   BB2_AS2.Stoerung.Res_24 := FALSE;
   BB2_AS2.Stoerung.Res_25 := FALSE;
   BB2_AS2.Stoerung.Res_26 := FALSE;
   BB2_AS2.Stoerung.Res_27 := FALSE;
   BB2_AS2.Stoerung.Res_28 := FALSE;
   BB2_AS2.Stoerung.Res_29 := FALSE;
   BB2_AS2.Stoerung.Res_30 := FALSE;
   BB2_AS2.Stoerung.Res_31 := FALSE;
   BB2_AS2.MW_I := 0.0;
   BB2_AS2.MW_P := 0.0;
   BB2_AS2.EZ := 0;
   BB2_AS2.BZ_akt := 27;
   BB2_AS2.BZ_ges := 978766;
   BB2_AS2.AZ_akt := 2137;
   BB2_AS2.ESH := 35306;
   BB2_AS2.SW_akt := 0.0;
   BB2_AS2.SW_Auto := 0.0;
   BB2_AS2.SW_out := 0.0;
   BB2_SR1.Status.Bed_vOrt := FALSE;
   BB2_SR1.Status.Bed_UV := FALSE;
   BB2_SR1.Status.Bed_NHV := FALSE;
   BB2_SR1.Status.Bed_PLS := TRUE;
   BB2_SR1.Status.BA_Hand := FALSE;
   BB2_SR1.Status.BA_Auto := TRUE;
   BB2_SR1.Status.RB_Ein1 := FALSE;
   BB2_SR1.Status.RB_Ein2 := FALSE;
   BB2_SR1.Status.RB_Aus := TRUE;
   BB2_SR1.Status.BFR_NS := FALSE;
   BB2_SR1.Status.BFR_ECS := FALSE;
   BB2_SR1.Status.BFR_ESK := FALSE;
   BB2_SR1.Status.BFR_MAZ := FALSE;
   BB2_SR1.Status.BFR_Rev := FALSE;
   BB2_SR1.Status.BFR_Ein1 := FALSE;
   BB2_SR1.Status.BFR_Ein2 := FALSE;
   BB2_SR1.Status.BM_Ein1 := FALSE;
   BB2_SR1.Status.BM_Ein2 := FALSE;
   BB2_SR1.Status.BM_Auf := FALSE;
   BB2_SR1.Status.BM_Zu := TRUE;
   BB2_SR1.Status.BM_Ein := FALSE;
   BB2_SR1.Status.BM_Aus := TRUE;
   BB2_SR1.Status.BM_Anst1 := FALSE;
   BB2_SR1.Status.BM_Anst2 := FALSE;
   BB2_SR1.Status.BM_Auto1 := FALSE;
   BB2_SR1.Status.BM_Auto2 := TRUE;
   BB2_SR1.Status.Res_26 := FALSE;
   BB2_SR1.Status.Res_27 := FALSE;
   BB2_SR1.Status.BB_NA := FALSE;
   BB2_SR1.Status.BB_AutoOk := TRUE;
   BB2_SR1.Status.BB_SS := FALSE;
   BB2_SR1.Status.BB_SSnq := FALSE;
   BB2_SR1.Stoerung.St_allg := FALSE;
   BB2_SR1.Stoerung.St_DMA := FALSE;
   BB2_SR1.Stoerung.St_DMZ := FALSE;
   BB2_SR1.Stoerung.St_FU := FALSE;
   BB2_SR1.Stoerung.St_TL := FALSE;
   BB2_SR1.Stoerung.St_UDr := FALSE;
   BB2_SR1.Stoerung.St_UeDr := FALSE;
   BB2_SR1.Stoerung.St_UeTemp := FALSE;
   BB2_SR1.Stoerung.St_Leck := FALSE;
   BB2_SR1.Stoerung.St_UeLM := FALSE;
   BB2_SR1.Stoerung.St_UeLE := FALSE;
   BB2_SR1.Stoerung.St_Kom_DP := FALSE;
   BB2_SR1.Stoerung.St_Kom_int := FALSE;
   BB2_SR1.Stoerung.St_int := FALSE;
   BB2_SR1.Stoerung.St_LZ := FALSE;
   BB2_SR1.Stoerung.St_BefLZ := FALSE;
   BB2_SR1.Stoerung.Wa_EZ := FALSE;
   BB2_SR1.Stoerung.Wa_Wart := FALSE;
   BB2_SR1.Stoerung.St_Strm := FALSE;
   BB2_SR1.Stoerung.Res_19 := FALSE;
   BB2_SR1.Stoerung.Res_20 := FALSE;
   BB2_SR1.Stoerung.Res_21 := FALSE;
   BB2_SR1.Stoerung.Res_22 := FALSE;
   BB2_SR1.Stoerung.Res_23 := FALSE;
   BB2_SR1.Stoerung.Res_24 := FALSE;
   BB2_SR1.Stoerung.Res_25 := FALSE;
   BB2_SR1.Stoerung.Res_26 := FALSE;
   BB2_SR1.Stoerung.Res_27 := FALSE;
   BB2_SR1.Stoerung.Res_28 := FALSE;
   BB2_SR1.Stoerung.Res_29 := FALSE;
   BB2_SR1.Stoerung.Res_30 := FALSE;
   BB2_SR1.Stoerung.Res_31 := FALSE;
   BB2_SR1.MW_I := 0.0;
   BB2_SR1.MW_P := 0.0;
   BB2_SR1.EZ := 0;
   BB2_SR1.BZ_akt := 179;
   BB2_SR1.BZ_ges := 3159816;
   BB2_SR1.AZ_akt := 5585;
   BB2_SR1.ESH := 17588;
   BB2_SR1.SW_akt := 0.0;
   BB2_SR1.SW_Auto := 0.0;
   BB2_SR1.SW_out := 0.0;
   BB2_SR2.Status.Bed_vOrt := FALSE;
   BB2_SR2.Status.Bed_UV := FALSE;
   BB2_SR2.Status.Bed_NHV := FALSE;
   BB2_SR2.Status.Bed_PLS := TRUE;
   BB2_SR2.Status.BA_Hand := FALSE;
   BB2_SR2.Status.BA_Auto := TRUE;
   BB2_SR2.Status.RB_Ein1 := FALSE;
   BB2_SR2.Status.RB_Ein2 := FALSE;
   BB2_SR2.Status.RB_Aus := TRUE;
   BB2_SR2.Status.BFR_NS := FALSE;
   BB2_SR2.Status.BFR_ECS := FALSE;
   BB2_SR2.Status.BFR_ESK := FALSE;
   BB2_SR2.Status.BFR_MAZ := FALSE;
   BB2_SR2.Status.BFR_Rev := FALSE;
   BB2_SR2.Status.BFR_Ein1 := FALSE;
   BB2_SR2.Status.BFR_Ein2 := FALSE;
   BB2_SR2.Status.BM_Ein1 := FALSE;
   BB2_SR2.Status.BM_Ein2 := FALSE;
   BB2_SR2.Status.BM_Auf := FALSE;
   BB2_SR2.Status.BM_Zu := TRUE;
   BB2_SR2.Status.BM_Ein := FALSE;
   BB2_SR2.Status.BM_Aus := TRUE;
   BB2_SR2.Status.BM_Anst1 := FALSE;
   BB2_SR2.Status.BM_Anst2 := FALSE;
   BB2_SR2.Status.BM_Auto1 := FALSE;
   BB2_SR2.Status.BM_Auto2 := TRUE;
   BB2_SR2.Status.Res_26 := FALSE;
   BB2_SR2.Status.Res_27 := FALSE;
   BB2_SR2.Status.BB_NA := FALSE;
   BB2_SR2.Status.BB_AutoOk := TRUE;
   BB2_SR2.Status.BB_SS := FALSE;
   BB2_SR2.Status.BB_SSnq := FALSE;
   BB2_SR2.Stoerung.St_allg := FALSE;
   BB2_SR2.Stoerung.St_DMA := FALSE;
   BB2_SR2.Stoerung.St_DMZ := FALSE;
   BB2_SR2.Stoerung.St_FU := FALSE;
   BB2_SR2.Stoerung.St_TL := FALSE;
   BB2_SR2.Stoerung.St_UDr := FALSE;
   BB2_SR2.Stoerung.St_UeDr := FALSE;
   BB2_SR2.Stoerung.St_UeTemp := FALSE;
   BB2_SR2.Stoerung.St_Leck := FALSE;
   BB2_SR2.Stoerung.St_UeLM := FALSE;
   BB2_SR2.Stoerung.St_UeLE := FALSE;
   BB2_SR2.Stoerung.St_Kom_DP := FALSE;
   BB2_SR2.Stoerung.St_Kom_int := FALSE;
   BB2_SR2.Stoerung.St_int := FALSE;
   BB2_SR2.Stoerung.St_LZ := FALSE;
   BB2_SR2.Stoerung.St_BefLZ := FALSE;
   BB2_SR2.Stoerung.Wa_EZ := FALSE;
   BB2_SR2.Stoerung.Wa_Wart := FALSE;
   BB2_SR2.Stoerung.St_Strm := FALSE;
   BB2_SR2.Stoerung.Res_19 := FALSE;
   BB2_SR2.Stoerung.Res_20 := FALSE;
   BB2_SR2.Stoerung.Res_21 := FALSE;
   BB2_SR2.Stoerung.Res_22 := FALSE;
   BB2_SR2.Stoerung.Res_23 := FALSE;
   BB2_SR2.Stoerung.Res_24 := FALSE;
   BB2_SR2.Stoerung.Res_25 := FALSE;
   BB2_SR2.Stoerung.Res_26 := FALSE;
   BB2_SR2.Stoerung.Res_27 := FALSE;
   BB2_SR2.Stoerung.Res_28 := FALSE;
   BB2_SR2.Stoerung.Res_29 := FALSE;
   BB2_SR2.Stoerung.Res_30 := FALSE;
   BB2_SR2.Stoerung.Res_31 := FALSE;
   BB2_SR2.MW_I := 0.0;
   BB2_SR2.MW_P := 0.0;
   BB2_SR2.EZ := 0;
   BB2_SR2.BZ_akt := 179;
   BB2_SR2.BZ_ges := 3129764;
   BB2_SR2.AZ_akt := 1985;
   BB2_SR2.ESH := 17409;
   BB2_SR2.SW_akt := 0.0;
   BB2_SR2.SW_Auto := 0.0;
   BB2_SR2.SW_out := 0.0;
   BB1_SR_K.Status.Bed_vOrt := FALSE;
   BB1_SR_K.Status.Bed_UV := FALSE;
   BB1_SR_K.Status.Bed_NHV := TRUE;
   BB1_SR_K.Status.Bed_PLS := FALSE;
   BB1_SR_K.Status.BA_Hand := FALSE;
   BB1_SR_K.Status.BA_Auto := TRUE;
   BB1_SR_K.Status.RB_Ein1 := FALSE;
   BB1_SR_K.Status.RB_Ein2 := FALSE;
   BB1_SR_K.Status.RB_Aus := TRUE;
   BB1_SR_K.Status.BFR_NS := FALSE;
   BB1_SR_K.Status.BFR_ECS := FALSE;
   BB1_SR_K.Status.BFR_ESK := FALSE;
   BB1_SR_K.Status.BFR_MAZ := FALSE;
   BB1_SR_K.Status.BFR_Rev := FALSE;
   BB1_SR_K.Status.BFR_Ein1 := FALSE;
   BB1_SR_K.Status.BFR_Ein2 := FALSE;
   BB1_SR_K.Status.BM_Ein1 := FALSE;
   BB1_SR_K.Status.BM_Ein2 := FALSE;
   BB1_SR_K.Status.BM_Auf := FALSE;
   BB1_SR_K.Status.BM_Zu := FALSE;
   BB1_SR_K.Status.BM_Ein := FALSE;
   BB1_SR_K.Status.BM_Aus := TRUE;
   BB1_SR_K.Status.BM_Anst1 := FALSE;
   BB1_SR_K.Status.BM_Anst2 := FALSE;
   BB1_SR_K.Status.BM_Auto1 := FALSE;
   BB1_SR_K.Status.BM_Auto2 := FALSE;
   BB1_SR_K.Status.Res_26 := FALSE;
   BB1_SR_K.Status.Res_27 := FALSE;
   BB1_SR_K.Status.BB_NA := FALSE;
   BB1_SR_K.Status.BB_AutoOk := FALSE;
   BB1_SR_K.Status.BB_SS := TRUE;
   BB1_SR_K.Status.BB_SSnq := FALSE;
   BB1_SR_K.Stoerung.St_allg := TRUE;
   BB1_SR_K.Stoerung.St_DMA := FALSE;
   BB1_SR_K.Stoerung.St_DMZ := FALSE;
   BB1_SR_K.Stoerung.St_FU := FALSE;
   BB1_SR_K.Stoerung.St_TL := FALSE;
   BB1_SR_K.Stoerung.St_UDr := FALSE;
   BB1_SR_K.Stoerung.St_UeDr := FALSE;
   BB1_SR_K.Stoerung.St_UeTemp := FALSE;
   BB1_SR_K.Stoerung.St_Leck := FALSE;
   BB1_SR_K.Stoerung.St_UeLM := FALSE;
   BB1_SR_K.Stoerung.St_UeLE := FALSE;
   BB1_SR_K.Stoerung.St_Kom_DP := FALSE;
   BB1_SR_K.Stoerung.St_Kom_int := FALSE;
   BB1_SR_K.Stoerung.St_int := FALSE;
   BB1_SR_K.Stoerung.St_LZ := FALSE;
   BB1_SR_K.Stoerung.St_BefLZ := FALSE;
   BB1_SR_K.Stoerung.Wa_EZ := FALSE;
   BB1_SR_K.Stoerung.Wa_Wart := FALSE;
   BB1_SR_K.Stoerung.St_Strm := FALSE;
   BB1_SR_K.Stoerung.Res_19 := FALSE;
   BB1_SR_K.Stoerung.Res_20 := FALSE;
   BB1_SR_K.Stoerung.Res_21 := FALSE;
   BB1_SR_K.Stoerung.Res_22 := FALSE;
   BB1_SR_K.Stoerung.Res_23 := FALSE;
   BB1_SR_K.Stoerung.Res_24 := FALSE;
   BB1_SR_K.Stoerung.Res_25 := FALSE;
   BB1_SR_K.Stoerung.Res_26 := FALSE;
   BB1_SR_K.Stoerung.Res_27 := FALSE;
   BB1_SR_K.Stoerung.Res_28 := FALSE;
   BB1_SR_K.Stoerung.Res_29 := FALSE;
   BB1_SR_K.Stoerung.Res_30 := FALSE;
   BB1_SR_K.Stoerung.Res_31 := FALSE;
   BB1_SR_K.MW_I := 0.0;
   BB1_SR_K.MW_P := 0.0;
   BB1_SR_K.EZ := 0;
   BB1_SR_K.BZ_akt := 180;
   BB1_SR_K.BZ_ges := 6365850;
   BB1_SR_K.AZ_akt := 2005;
   BB1_SR_K.ESH := 34998;
   BB1_SR_K.SW_akt := 0.0;
   BB1_SR_K.SW_Auto := 0.0;
   BB1_SR_K.SW_out := 0.0;
   Zulauf_AR_P1.Status.Bed_vOrt := FALSE;
   Zulauf_AR_P1.Status.Bed_UV := FALSE;
   Zulauf_AR_P1.Status.Bed_NHV := TRUE;
   Zulauf_AR_P1.Status.Bed_PLS := FALSE;
   Zulauf_AR_P1.Status.BA_Hand := FALSE;
   Zulauf_AR_P1.Status.BA_Auto := TRUE;
   Zulauf_AR_P1.Status.RB_Ein1 := FALSE;
   Zulauf_AR_P1.Status.RB_Ein2 := FALSE;
   Zulauf_AR_P1.Status.RB_Aus := TRUE;
   Zulauf_AR_P1.Status.BFR_NS := FALSE;
   Zulauf_AR_P1.Status.BFR_ECS := FALSE;
   Zulauf_AR_P1.Status.BFR_ESK := FALSE;
   Zulauf_AR_P1.Status.BFR_MAZ := FALSE;
   Zulauf_AR_P1.Status.BFR_Rev := FALSE;
   Zulauf_AR_P1.Status.BFR_Ein1 := FALSE;
   Zulauf_AR_P1.Status.BFR_Ein2 := FALSE;
   Zulauf_AR_P1.Status.BM_Ein1 := FALSE;
   Zulauf_AR_P1.Status.BM_Ein2 := FALSE;
   Zulauf_AR_P1.Status.BM_Auf := FALSE;
   Zulauf_AR_P1.Status.BM_Zu := FALSE;
   Zulauf_AR_P1.Status.BM_Ein := FALSE;
   Zulauf_AR_P1.Status.BM_Aus := TRUE;
   Zulauf_AR_P1.Status.BM_Anst1 := FALSE;
   Zulauf_AR_P1.Status.BM_Anst2 := FALSE;
   Zulauf_AR_P1.Status.BM_Auto1 := FALSE;
   Zulauf_AR_P1.Status.BM_Auto2 := FALSE;
   Zulauf_AR_P1.Status.Res_26 := FALSE;
   Zulauf_AR_P1.Status.Res_27 := FALSE;
   Zulauf_AR_P1.Status.BB_NA := FALSE;
   Zulauf_AR_P1.Status.BB_AutoOk := TRUE;
   Zulauf_AR_P1.Status.BB_SS := FALSE;
   Zulauf_AR_P1.Status.BB_SSnq := FALSE;
   Zulauf_AR_P1.Stoerung.St_allg := FALSE;
   Zulauf_AR_P1.Stoerung.St_DMA := FALSE;
   Zulauf_AR_P1.Stoerung.St_DMZ := FALSE;
   Zulauf_AR_P1.Stoerung.St_FU := FALSE;
   Zulauf_AR_P1.Stoerung.St_TL := FALSE;
   Zulauf_AR_P1.Stoerung.St_UDr := FALSE;
   Zulauf_AR_P1.Stoerung.St_UeDr := FALSE;
   Zulauf_AR_P1.Stoerung.St_UeTemp := FALSE;
   Zulauf_AR_P1.Stoerung.St_Leck := FALSE;
   Zulauf_AR_P1.Stoerung.St_UeLM := FALSE;
   Zulauf_AR_P1.Stoerung.St_UeLE := FALSE;
   Zulauf_AR_P1.Stoerung.St_Kom_DP := FALSE;
   Zulauf_AR_P1.Stoerung.St_Kom_int := FALSE;
   Zulauf_AR_P1.Stoerung.St_int := FALSE;
   Zulauf_AR_P1.Stoerung.St_LZ := FALSE;
   Zulauf_AR_P1.Stoerung.St_BefLZ := FALSE;
   Zulauf_AR_P1.Stoerung.Wa_EZ := FALSE;
   Zulauf_AR_P1.Stoerung.Wa_Wart := FALSE;
   Zulauf_AR_P1.Stoerung.St_Strm := FALSE;
   Zulauf_AR_P1.Stoerung.Res_19 := FALSE;
   Zulauf_AR_P1.Stoerung.Res_20 := FALSE;
   Zulauf_AR_P1.Stoerung.Res_21 := FALSE;
   Zulauf_AR_P1.Stoerung.Res_22 := FALSE;
   Zulauf_AR_P1.Stoerung.Res_23 := FALSE;
   Zulauf_AR_P1.Stoerung.Res_24 := FALSE;
   Zulauf_AR_P1.Stoerung.Res_25 := FALSE;
   Zulauf_AR_P1.Stoerung.Res_26 := FALSE;
   Zulauf_AR_P1.Stoerung.Res_27 := FALSE;
   Zulauf_AR_P1.Stoerung.Res_28 := FALSE;
   Zulauf_AR_P1.Stoerung.Res_29 := FALSE;
   Zulauf_AR_P1.Stoerung.Res_30 := FALSE;
   Zulauf_AR_P1.Stoerung.Res_31 := FALSE;
   Zulauf_AR_P1.MW_I := 0.0;
   Zulauf_AR_P1.MW_P := 0.0;
   Zulauf_AR_P1.EZ := 0;
   Zulauf_AR_P1.BZ_akt := 0;
   Zulauf_AR_P1.BZ_ges := 0;
   Zulauf_AR_P1.AZ_akt := 132_442_977;
   Zulauf_AR_P1.ESH := 0;
   Zulauf_AR_P1.SW_akt := 0.0;
   Zulauf_AR_P1.SW_Auto := 0.0;
   Zulauf_AR_P1.SW_out := 0.0;
   Zulauf_AR_P2.Status.Bed_vOrt := FALSE;
   Zulauf_AR_P2.Status.Bed_UV := FALSE;
   Zulauf_AR_P2.Status.Bed_NHV := TRUE;
   Zulauf_AR_P2.Status.Bed_PLS := FALSE;
   Zulauf_AR_P2.Status.BA_Hand := FALSE;
   Zulauf_AR_P2.Status.BA_Auto := TRUE;
   Zulauf_AR_P2.Status.RB_Ein1 := FALSE;
   Zulauf_AR_P2.Status.RB_Ein2 := FALSE;
   Zulauf_AR_P2.Status.RB_Aus := TRUE;
   Zulauf_AR_P2.Status.BFR_NS := FALSE;
   Zulauf_AR_P2.Status.BFR_ECS := FALSE;
   Zulauf_AR_P2.Status.BFR_ESK := FALSE;
   Zulauf_AR_P2.Status.BFR_MAZ := FALSE;
   Zulauf_AR_P2.Status.BFR_Rev := FALSE;
   Zulauf_AR_P2.Status.BFR_Ein1 := FALSE;
   Zulauf_AR_P2.Status.BFR_Ein2 := FALSE;
   Zulauf_AR_P2.Status.BM_Ein1 := FALSE;
   Zulauf_AR_P2.Status.BM_Ein2 := FALSE;
   Zulauf_AR_P2.Status.BM_Auf := FALSE;
   Zulauf_AR_P2.Status.BM_Zu := FALSE;
   Zulauf_AR_P2.Status.BM_Ein := FALSE;
   Zulauf_AR_P2.Status.BM_Aus := TRUE;
   Zulauf_AR_P2.Status.BM_Anst1 := FALSE;
   Zulauf_AR_P2.Status.BM_Anst2 := FALSE;
   Zulauf_AR_P2.Status.BM_Auto1 := FALSE;
   Zulauf_AR_P2.Status.BM_Auto2 := FALSE;
   Zulauf_AR_P2.Status.Res_26 := FALSE;
   Zulauf_AR_P2.Status.Res_27 := FALSE;
   Zulauf_AR_P2.Status.BB_NA := FALSE;
   Zulauf_AR_P2.Status.BB_AutoOk := TRUE;
   Zulauf_AR_P2.Status.BB_SS := FALSE;
   Zulauf_AR_P2.Status.BB_SSnq := FALSE;
   Zulauf_AR_P2.Stoerung.St_allg := FALSE;
   Zulauf_AR_P2.Stoerung.St_DMA := FALSE;
   Zulauf_AR_P2.Stoerung.St_DMZ := FALSE;
   Zulauf_AR_P2.Stoerung.St_FU := FALSE;
   Zulauf_AR_P2.Stoerung.St_TL := FALSE;
   Zulauf_AR_P2.Stoerung.St_UDr := FALSE;
   Zulauf_AR_P2.Stoerung.St_UeDr := FALSE;
   Zulauf_AR_P2.Stoerung.St_UeTemp := FALSE;
   Zulauf_AR_P2.Stoerung.St_Leck := FALSE;
   Zulauf_AR_P2.Stoerung.St_UeLM := FALSE;
   Zulauf_AR_P2.Stoerung.St_UeLE := FALSE;
   Zulauf_AR_P2.Stoerung.St_Kom_DP := FALSE;
   Zulauf_AR_P2.Stoerung.St_Kom_int := FALSE;
   Zulauf_AR_P2.Stoerung.St_int := FALSE;
   Zulauf_AR_P2.Stoerung.St_LZ := FALSE;
   Zulauf_AR_P2.Stoerung.St_BefLZ := FALSE;
   Zulauf_AR_P2.Stoerung.Wa_EZ := FALSE;
   Zulauf_AR_P2.Stoerung.Wa_Wart := FALSE;
   Zulauf_AR_P2.Stoerung.St_Strm := FALSE;
   Zulauf_AR_P2.Stoerung.Res_19 := FALSE;
   Zulauf_AR_P2.Stoerung.Res_20 := FALSE;
   Zulauf_AR_P2.Stoerung.Res_21 := FALSE;
   Zulauf_AR_P2.Stoerung.Res_22 := FALSE;
   Zulauf_AR_P2.Stoerung.Res_23 := FALSE;
   Zulauf_AR_P2.Stoerung.Res_24 := FALSE;
   Zulauf_AR_P2.Stoerung.Res_25 := FALSE;
   Zulauf_AR_P2.Stoerung.Res_26 := FALSE;
   Zulauf_AR_P2.Stoerung.Res_27 := FALSE;
   Zulauf_AR_P2.Stoerung.Res_28 := FALSE;
   Zulauf_AR_P2.Stoerung.Res_29 := FALSE;
   Zulauf_AR_P2.Stoerung.Res_30 := FALSE;
   Zulauf_AR_P2.Stoerung.Res_31 := FALSE;
   Zulauf_AR_P2.MW_I := 0.0;
   Zulauf_AR_P2.MW_P := 0.0;
   Zulauf_AR_P2.EZ := 0;
   Zulauf_AR_P2.BZ_akt := 676;
   Zulauf_AR_P2.BZ_ges := 676;
   Zulauf_AR_P2.AZ_akt := 132_196_371;
   Zulauf_AR_P2.ESH := 1;
   Zulauf_AR_P2.SW_akt := 0.0;
   Zulauf_AR_P2.SW_Auto := 0.0;
   Zulauf_AR_P2.SW_out := 0.0;
   Zulauf_AS.Status.Bed_vOrt := FALSE;
   Zulauf_AS.Status.Bed_UV := FALSE;
   Zulauf_AS.Status.Bed_NHV := TRUE;
   Zulauf_AS.Status.Bed_PLS := FALSE;
   Zulauf_AS.Status.BA_Hand := FALSE;
   Zulauf_AS.Status.BA_Auto := TRUE;
   Zulauf_AS.Status.RB_Ein1 := FALSE;
   Zulauf_AS.Status.RB_Ein2 := FALSE;
   Zulauf_AS.Status.RB_Aus := TRUE;
   Zulauf_AS.Status.BFR_NS := FALSE;
   Zulauf_AS.Status.BFR_ECS := FALSE;
   Zulauf_AS.Status.BFR_ESK := FALSE;
   Zulauf_AS.Status.BFR_MAZ := FALSE;
   Zulauf_AS.Status.BFR_Rev := FALSE;
   Zulauf_AS.Status.BFR_Ein1 := FALSE;
   Zulauf_AS.Status.BFR_Ein2 := FALSE;
   Zulauf_AS.Status.BM_Ein1 := FALSE;
   Zulauf_AS.Status.BM_Ein2 := FALSE;
   Zulauf_AS.Status.BM_Auf := FALSE;
   Zulauf_AS.Status.BM_Zu := FALSE;
   Zulauf_AS.Status.BM_Ein := FALSE;
   Zulauf_AS.Status.BM_Aus := TRUE;
   Zulauf_AS.Status.BM_Anst1 := FALSE;
   Zulauf_AS.Status.BM_Anst2 := FALSE;
   Zulauf_AS.Status.BM_Auto1 := FALSE;
   Zulauf_AS.Status.BM_Auto2 := FALSE;
   Zulauf_AS.Status.Res_26 := FALSE;
   Zulauf_AS.Status.Res_27 := FALSE;
   Zulauf_AS.Status.BB_NA := FALSE;
   Zulauf_AS.Status.BB_AutoOk := FALSE;
   Zulauf_AS.Status.BB_SS := TRUE;
   Zulauf_AS.Status.BB_SSnq := TRUE;
   Zulauf_AS.Stoerung.St_allg := TRUE;
   Zulauf_AS.Stoerung.St_DMA := FALSE;
   Zulauf_AS.Stoerung.St_DMZ := FALSE;
   Zulauf_AS.Stoerung.St_FU := FALSE;
   Zulauf_AS.Stoerung.St_TL := FALSE;
   Zulauf_AS.Stoerung.St_UDr := FALSE;
   Zulauf_AS.Stoerung.St_UeDr := FALSE;
   Zulauf_AS.Stoerung.St_UeTemp := FALSE;
   Zulauf_AS.Stoerung.St_Leck := FALSE;
   Zulauf_AS.Stoerung.St_UeLM := FALSE;
   Zulauf_AS.Stoerung.St_UeLE := FALSE;
   Zulauf_AS.Stoerung.St_Kom_DP := FALSE;
   Zulauf_AS.Stoerung.St_Kom_int := FALSE;
   Zulauf_AS.Stoerung.St_int := FALSE;
   Zulauf_AS.Stoerung.St_LZ := FALSE;
   Zulauf_AS.Stoerung.St_BefLZ := FALSE;
   Zulauf_AS.Stoerung.Wa_EZ := FALSE;
   Zulauf_AS.Stoerung.Wa_Wart := FALSE;
   Zulauf_AS.Stoerung.St_Strm := FALSE;
   Zulauf_AS.Stoerung.Res_19 := FALSE;
   Zulauf_AS.Stoerung.Res_20 := FALSE;
   Zulauf_AS.Stoerung.Res_21 := FALSE;
   Zulauf_AS.Stoerung.Res_22 := FALSE;
   Zulauf_AS.Stoerung.Res_23 := FALSE;
   Zulauf_AS.Stoerung.Res_24 := FALSE;
   Zulauf_AS.Stoerung.Res_25 := FALSE;
   Zulauf_AS.Stoerung.Res_26 := FALSE;
   Zulauf_AS.Stoerung.Res_27 := FALSE;
   Zulauf_AS.Stoerung.Res_28 := FALSE;
   Zulauf_AS.Stoerung.Res_29 := FALSE;
   Zulauf_AS.Stoerung.Res_30 := FALSE;
   Zulauf_AS.Stoerung.Res_31 := FALSE;
   Zulauf_AS.MW_I := 0.0;
   Zulauf_AS.MW_P := 0.0;
   Zulauf_AS.EZ := 0;
   Zulauf_AS.BZ_akt := 0;
   Zulauf_AS.BZ_ges := 0;
   Zulauf_AS.AZ_akt := 132_442_977;
   Zulauf_AS.ESH := 0;
   Zulauf_AS.SW_akt := 0.0;
   Zulauf_AS.SW_Auto := 0.0;
   Zulauf_AS.SW_out := 0.0;
   Zulauf_RA_SA.Status.Bed_vOrt := FALSE;
   Zulauf_RA_SA.Status.Bed_UV := FALSE;
   Zulauf_RA_SA.Status.Bed_NHV := TRUE;
   Zulauf_RA_SA.Status.Bed_PLS := FALSE;
   Zulauf_RA_SA.Status.BA_Hand := FALSE;
   Zulauf_RA_SA.Status.BA_Auto := TRUE;
   Zulauf_RA_SA.Status.RB_Ein1 := FALSE;
   Zulauf_RA_SA.Status.RB_Ein2 := FALSE;
   Zulauf_RA_SA.Status.RB_Aus := TRUE;
   Zulauf_RA_SA.Status.BFR_NS := FALSE;
   Zulauf_RA_SA.Status.BFR_ECS := FALSE;
   Zulauf_RA_SA.Status.BFR_ESK := FALSE;
   Zulauf_RA_SA.Status.BFR_MAZ := FALSE;
   Zulauf_RA_SA.Status.BFR_Rev := FALSE;
   Zulauf_RA_SA.Status.BFR_Ein1 := FALSE;
   Zulauf_RA_SA.Status.BFR_Ein2 := FALSE;
   Zulauf_RA_SA.Status.BM_Ein1 := FALSE;
   Zulauf_RA_SA.Status.BM_Ein2 := FALSE;
   Zulauf_RA_SA.Status.BM_Auf := FALSE;
   Zulauf_RA_SA.Status.BM_Zu := FALSE;
   Zulauf_RA_SA.Status.BM_Ein := FALSE;
   Zulauf_RA_SA.Status.BM_Aus := TRUE;
   Zulauf_RA_SA.Status.BM_Anst1 := FALSE;
   Zulauf_RA_SA.Status.BM_Anst2 := FALSE;
   Zulauf_RA_SA.Status.BM_Auto1 := FALSE;
   Zulauf_RA_SA.Status.BM_Auto2 := FALSE;
   Zulauf_RA_SA.Status.Res_26 := FALSE;
   Zulauf_RA_SA.Status.Res_27 := FALSE;
   Zulauf_RA_SA.Status.BB_NA := FALSE;
   Zulauf_RA_SA.Status.BB_AutoOk := TRUE;
   Zulauf_RA_SA.Status.BB_SS := FALSE;
   Zulauf_RA_SA.Status.BB_SSnq := FALSE;
   Zulauf_RA_SA.Stoerung.St_allg := FALSE;
   Zulauf_RA_SA.Stoerung.St_DMA := FALSE;
   Zulauf_RA_SA.Stoerung.St_DMZ := FALSE;
   Zulauf_RA_SA.Stoerung.St_FU := FALSE;
   Zulauf_RA_SA.Stoerung.St_TL := FALSE;
   Zulauf_RA_SA.Stoerung.St_UDr := FALSE;
   Zulauf_RA_SA.Stoerung.St_UeDr := FALSE;
   Zulauf_RA_SA.Stoerung.St_UeTemp := FALSE;
   Zulauf_RA_SA.Stoerung.St_Leck := FALSE;
   Zulauf_RA_SA.Stoerung.St_UeLM := FALSE;
   Zulauf_RA_SA.Stoerung.St_UeLE := FALSE;
   Zulauf_RA_SA.Stoerung.St_Kom_DP := FALSE;
   Zulauf_RA_SA.Stoerung.St_Kom_int := FALSE;
   Zulauf_RA_SA.Stoerung.St_int := FALSE;
   Zulauf_RA_SA.Stoerung.St_LZ := FALSE;
   Zulauf_RA_SA.Stoerung.St_BefLZ := FALSE;
   Zulauf_RA_SA.Stoerung.Wa_EZ := FALSE;
   Zulauf_RA_SA.Stoerung.Wa_Wart := FALSE;
   Zulauf_RA_SA.Stoerung.St_Strm := FALSE;
   Zulauf_RA_SA.Stoerung.Res_19 := FALSE;
   Zulauf_RA_SA.Stoerung.Res_20 := FALSE;
   Zulauf_RA_SA.Stoerung.Res_21 := FALSE;
   Zulauf_RA_SA.Stoerung.Res_22 := FALSE;
   Zulauf_RA_SA.Stoerung.Res_23 := FALSE;
   Zulauf_RA_SA.Stoerung.Res_24 := FALSE;
   Zulauf_RA_SA.Stoerung.Res_25 := FALSE;
   Zulauf_RA_SA.Stoerung.Res_26 := FALSE;
   Zulauf_RA_SA.Stoerung.Res_27 := FALSE;
   Zulauf_RA_SA.Stoerung.Res_28 := FALSE;
   Zulauf_RA_SA.Stoerung.Res_29 := FALSE;
   Zulauf_RA_SA.Stoerung.Res_30 := FALSE;
   Zulauf_RA_SA.Stoerung.Res_31 := FALSE;
   Zulauf_RA_SA.MW_I := 0.0;
   Zulauf_RA_SA.MW_P := 0.0;
   Zulauf_RA_SA.EZ := 0;
   Zulauf_RA_SA.BZ_akt := 29;
   Zulauf_RA_SA.BZ_ges := 72610;
   Zulauf_RA_SA.AZ_akt := 35;
   Zulauf_RA_SA.ESH := 2460;
   Zulauf_RA_SA.SW_akt := 0.0;
   Zulauf_RA_SA.SW_Auto := 0.0;
   Zulauf_RA_SA.SW_out := 0.0;
   Zulauf_RA_HZS.Status.Bed_vOrt := FALSE;
   Zulauf_RA_HZS.Status.Bed_UV := FALSE;
   Zulauf_RA_HZS.Status.Bed_NHV := TRUE;
   Zulauf_RA_HZS.Status.Bed_PLS := FALSE;
   Zulauf_RA_HZS.Status.BA_Hand := FALSE;
   Zulauf_RA_HZS.Status.BA_Auto := TRUE;
   Zulauf_RA_HZS.Status.RB_Ein1 := FALSE;
   Zulauf_RA_HZS.Status.RB_Ein2 := FALSE;
   Zulauf_RA_HZS.Status.RB_Aus := TRUE;
   Zulauf_RA_HZS.Status.BFR_NS := FALSE;
   Zulauf_RA_HZS.Status.BFR_ECS := FALSE;
   Zulauf_RA_HZS.Status.BFR_ESK := FALSE;
   Zulauf_RA_HZS.Status.BFR_MAZ := FALSE;
   Zulauf_RA_HZS.Status.BFR_Rev := FALSE;
   Zulauf_RA_HZS.Status.BFR_Ein1 := FALSE;
   Zulauf_RA_HZS.Status.BFR_Ein2 := FALSE;
   Zulauf_RA_HZS.Status.BM_Ein1 := FALSE;
   Zulauf_RA_HZS.Status.BM_Ein2 := FALSE;
   Zulauf_RA_HZS.Status.BM_Auf := FALSE;
   Zulauf_RA_HZS.Status.BM_Zu := FALSE;
   Zulauf_RA_HZS.Status.BM_Ein := FALSE;
   Zulauf_RA_HZS.Status.BM_Aus := TRUE;
   Zulauf_RA_HZS.Status.BM_Anst1 := FALSE;
   Zulauf_RA_HZS.Status.BM_Anst2 := FALSE;
   Zulauf_RA_HZS.Status.BM_Auto1 := FALSE;
   Zulauf_RA_HZS.Status.BM_Auto2 := FALSE;
   Zulauf_RA_HZS.Status.Res_26 := FALSE;
   Zulauf_RA_HZS.Status.Res_27 := FALSE;
   Zulauf_RA_HZS.Status.BB_NA := FALSE;
   Zulauf_RA_HZS.Status.BB_AutoOk := TRUE;
   Zulauf_RA_HZS.Status.BB_SS := FALSE;
   Zulauf_RA_HZS.Status.BB_SSnq := FALSE;
   Zulauf_RA_HZS.Stoerung.St_allg := FALSE;
   Zulauf_RA_HZS.Stoerung.St_DMA := FALSE;
   Zulauf_RA_HZS.Stoerung.St_DMZ := FALSE;
   Zulauf_RA_HZS.Stoerung.St_FU := FALSE;
   Zulauf_RA_HZS.Stoerung.St_TL := FALSE;
   Zulauf_RA_HZS.Stoerung.St_UDr := FALSE;
   Zulauf_RA_HZS.Stoerung.St_UeDr := FALSE;
   Zulauf_RA_HZS.Stoerung.St_UeTemp := FALSE;
   Zulauf_RA_HZS.Stoerung.St_Leck := FALSE;
   Zulauf_RA_HZS.Stoerung.St_UeLM := FALSE;
   Zulauf_RA_HZS.Stoerung.St_UeLE := FALSE;
   Zulauf_RA_HZS.Stoerung.St_Kom_DP := FALSE;
   Zulauf_RA_HZS.Stoerung.St_Kom_int := FALSE;
   Zulauf_RA_HZS.Stoerung.St_int := FALSE;
   Zulauf_RA_HZS.Stoerung.St_LZ := FALSE;
   Zulauf_RA_HZS.Stoerung.St_BefLZ := FALSE;
   Zulauf_RA_HZS.Stoerung.Wa_EZ := FALSE;
   Zulauf_RA_HZS.Stoerung.Wa_Wart := FALSE;
   Zulauf_RA_HZS.Stoerung.St_Strm := FALSE;
   Zulauf_RA_HZS.Stoerung.Res_19 := FALSE;
   Zulauf_RA_HZS.Stoerung.Res_20 := FALSE;
   Zulauf_RA_HZS.Stoerung.Res_21 := FALSE;
   Zulauf_RA_HZS.Stoerung.Res_22 := FALSE;
   Zulauf_RA_HZS.Stoerung.Res_23 := FALSE;
   Zulauf_RA_HZS.Stoerung.Res_24 := FALSE;
   Zulauf_RA_HZS.Stoerung.Res_25 := FALSE;
   Zulauf_RA_HZS.Stoerung.Res_26 := FALSE;
   Zulauf_RA_HZS.Stoerung.Res_27 := FALSE;
   Zulauf_RA_HZS.Stoerung.Res_28 := FALSE;
   Zulauf_RA_HZS.Stoerung.Res_29 := FALSE;
   Zulauf_RA_HZS.Stoerung.Res_30 := FALSE;
   Zulauf_RA_HZS.Stoerung.Res_31 := FALSE;
   Zulauf_RA_HZS.MW_I := 0.0;
   Zulauf_RA_HZS.MW_P := 0.0;
   Zulauf_RA_HZS.EZ := 0;
   Zulauf_RA_HZS.BZ_akt := 12;
   Zulauf_RA_HZS.BZ_ges := 15965;
   Zulauf_RA_HZS.AZ_akt := 519;
   Zulauf_RA_HZS.ESH := 1345;
   Zulauf_RA_HZS.SW_akt := 0.0;
   Zulauf_RA_HZS.SW_Auto := 0.0;
   Zulauf_RA_HZS.SW_out := 0.0;
   Zulauf_RA_VKS.Status.Bed_vOrt := FALSE;
   Zulauf_RA_VKS.Status.Bed_UV := FALSE;
   Zulauf_RA_VKS.Status.Bed_NHV := TRUE;
   Zulauf_RA_VKS.Status.Bed_PLS := FALSE;
   Zulauf_RA_VKS.Status.BA_Hand := FALSE;
   Zulauf_RA_VKS.Status.BA_Auto := TRUE;
   Zulauf_RA_VKS.Status.RB_Ein1 := FALSE;
   Zulauf_RA_VKS.Status.RB_Ein2 := FALSE;
   Zulauf_RA_VKS.Status.RB_Aus := TRUE;
   Zulauf_RA_VKS.Status.BFR_NS := FALSE;
   Zulauf_RA_VKS.Status.BFR_ECS := FALSE;
   Zulauf_RA_VKS.Status.BFR_ESK := FALSE;
   Zulauf_RA_VKS.Status.BFR_MAZ := FALSE;
   Zulauf_RA_VKS.Status.BFR_Rev := FALSE;
   Zulauf_RA_VKS.Status.BFR_Ein1 := FALSE;
   Zulauf_RA_VKS.Status.BFR_Ein2 := FALSE;
   Zulauf_RA_VKS.Status.BM_Ein1 := FALSE;
   Zulauf_RA_VKS.Status.BM_Ein2 := FALSE;
   Zulauf_RA_VKS.Status.BM_Auf := FALSE;
   Zulauf_RA_VKS.Status.BM_Zu := FALSE;
   Zulauf_RA_VKS.Status.BM_Ein := FALSE;
   Zulauf_RA_VKS.Status.BM_Aus := TRUE;
   Zulauf_RA_VKS.Status.BM_Anst1 := FALSE;
   Zulauf_RA_VKS.Status.BM_Anst2 := FALSE;
   Zulauf_RA_VKS.Status.BM_Auto1 := FALSE;
   Zulauf_RA_VKS.Status.BM_Auto2 := FALSE;
   Zulauf_RA_VKS.Status.Res_26 := FALSE;
   Zulauf_RA_VKS.Status.Res_27 := FALSE;
   Zulauf_RA_VKS.Status.BB_NA := FALSE;
   Zulauf_RA_VKS.Status.BB_AutoOk := TRUE;
   Zulauf_RA_VKS.Status.BB_SS := FALSE;
   Zulauf_RA_VKS.Status.BB_SSnq := FALSE;
   Zulauf_RA_VKS.Stoerung.St_allg := FALSE;
   Zulauf_RA_VKS.Stoerung.St_DMA := FALSE;
   Zulauf_RA_VKS.Stoerung.St_DMZ := FALSE;
   Zulauf_RA_VKS.Stoerung.St_FU := FALSE;
   Zulauf_RA_VKS.Stoerung.St_TL := FALSE;
   Zulauf_RA_VKS.Stoerung.St_UDr := FALSE;
   Zulauf_RA_VKS.Stoerung.St_UeDr := FALSE;
   Zulauf_RA_VKS.Stoerung.St_UeTemp := FALSE;
   Zulauf_RA_VKS.Stoerung.St_Leck := FALSE;
   Zulauf_RA_VKS.Stoerung.St_UeLM := FALSE;
   Zulauf_RA_VKS.Stoerung.St_UeLE := FALSE;
   Zulauf_RA_VKS.Stoerung.St_Kom_DP := FALSE;
   Zulauf_RA_VKS.Stoerung.St_Kom_int := FALSE;
   Zulauf_RA_VKS.Stoerung.St_int := FALSE;
   Zulauf_RA_VKS.Stoerung.St_LZ := FALSE;
   Zulauf_RA_VKS.Stoerung.St_BefLZ := FALSE;
   Zulauf_RA_VKS.Stoerung.Wa_EZ := FALSE;
   Zulauf_RA_VKS.Stoerung.Wa_Wart := FALSE;
   Zulauf_RA_VKS.Stoerung.St_Strm := FALSE;
   Zulauf_RA_VKS.Stoerung.Res_19 := FALSE;
   Zulauf_RA_VKS.Stoerung.Res_20 := FALSE;
   Zulauf_RA_VKS.Stoerung.Res_21 := FALSE;
   Zulauf_RA_VKS.Stoerung.Res_22 := FALSE;
   Zulauf_RA_VKS.Stoerung.Res_23 := FALSE;
   Zulauf_RA_VKS.Stoerung.Res_24 := FALSE;
   Zulauf_RA_VKS.Stoerung.Res_25 := FALSE;
   Zulauf_RA_VKS.Stoerung.Res_26 := FALSE;
   Zulauf_RA_VKS.Stoerung.Res_27 := FALSE;
   Zulauf_RA_VKS.Stoerung.Res_28 := FALSE;
   Zulauf_RA_VKS.Stoerung.Res_29 := FALSE;
   Zulauf_RA_VKS.Stoerung.Res_30 := FALSE;
   Zulauf_RA_VKS.Stoerung.Res_31 := FALSE;
   Zulauf_RA_VKS.MW_I := 0.0;
   Zulauf_RA_VKS.MW_P := 0.0;
   Zulauf_RA_VKS.EZ := 0;
   Zulauf_RA_VKS.BZ_akt := 17;
   Zulauf_RA_VKS.BZ_ges := 23886;
   Zulauf_RA_VKS.AZ_akt := 514;
   Zulauf_RA_VKS.ESH := 1347;
   Zulauf_RA_VKS.SW_akt := 0.0;
   Zulauf_RA_VKS.SW_Auto := 0.0;
   Zulauf_RA_VKS.SW_out := 0.0;
   Zulauf_RA_V.Status.Bed_vOrt := FALSE;
   Zulauf_RA_V.Status.Bed_UV := FALSE;
   Zulauf_RA_V.Status.Bed_NHV := TRUE;
   Zulauf_RA_V.Status.Bed_PLS := FALSE;
   Zulauf_RA_V.Status.BA_Hand := FALSE;
   Zulauf_RA_V.Status.BA_Auto := TRUE;
   Zulauf_RA_V.Status.RB_Ein1 := TRUE;
   Zulauf_RA_V.Status.RB_Ein2 := FALSE;
   Zulauf_RA_V.Status.RB_Aus := FALSE;
   Zulauf_RA_V.Status.BFR_NS := FALSE;
   Zulauf_RA_V.Status.BFR_ECS := FALSE;
   Zulauf_RA_V.Status.BFR_ESK := FALSE;
   Zulauf_RA_V.Status.BFR_MAZ := FALSE;
   Zulauf_RA_V.Status.BFR_Rev := FALSE;
   Zulauf_RA_V.Status.BFR_Ein1 := FALSE;
   Zulauf_RA_V.Status.BFR_Ein2 := FALSE;
   Zulauf_RA_V.Status.BM_Ein1 := TRUE;
   Zulauf_RA_V.Status.BM_Ein2 := FALSE;
   Zulauf_RA_V.Status.BM_Auf := FALSE;
   Zulauf_RA_V.Status.BM_Zu := FALSE;
   Zulauf_RA_V.Status.BM_Ein := TRUE;
   Zulauf_RA_V.Status.BM_Aus := FALSE;
   Zulauf_RA_V.Status.BM_Anst1 := FALSE;
   Zulauf_RA_V.Status.BM_Anst2 := FALSE;
   Zulauf_RA_V.Status.BM_Auto1 := FALSE;
   Zulauf_RA_V.Status.BM_Auto2 := FALSE;
   Zulauf_RA_V.Status.Res_26 := FALSE;
   Zulauf_RA_V.Status.Res_27 := FALSE;
   Zulauf_RA_V.Status.BB_NA := FALSE;
   Zulauf_RA_V.Status.BB_AutoOk := TRUE;
   Zulauf_RA_V.Status.BB_SS := FALSE;
   Zulauf_RA_V.Status.BB_SSnq := FALSE;
   Zulauf_RA_V.Stoerung.St_allg := FALSE;
   Zulauf_RA_V.Stoerung.St_DMA := FALSE;
   Zulauf_RA_V.Stoerung.St_DMZ := FALSE;
   Zulauf_RA_V.Stoerung.St_FU := FALSE;
   Zulauf_RA_V.Stoerung.St_TL := FALSE;
   Zulauf_RA_V.Stoerung.St_UDr := FALSE;
   Zulauf_RA_V.Stoerung.St_UeDr := FALSE;
   Zulauf_RA_V.Stoerung.St_UeTemp := FALSE;
   Zulauf_RA_V.Stoerung.St_Leck := FALSE;
   Zulauf_RA_V.Stoerung.St_UeLM := FALSE;
   Zulauf_RA_V.Stoerung.St_UeLE := FALSE;
   Zulauf_RA_V.Stoerung.St_Kom_DP := FALSE;
   Zulauf_RA_V.Stoerung.St_Kom_int := FALSE;
   Zulauf_RA_V.Stoerung.St_int := FALSE;
   Zulauf_RA_V.Stoerung.St_LZ := FALSE;
   Zulauf_RA_V.Stoerung.St_BefLZ := FALSE;
   Zulauf_RA_V.Stoerung.Wa_EZ := FALSE;
   Zulauf_RA_V.Stoerung.Wa_Wart := FALSE;
   Zulauf_RA_V.Stoerung.St_Strm := FALSE;
   Zulauf_RA_V.Stoerung.Res_19 := FALSE;
   Zulauf_RA_V.Stoerung.Res_20 := FALSE;
   Zulauf_RA_V.Stoerung.Res_21 := FALSE;
   Zulauf_RA_V.Stoerung.Res_22 := FALSE;
   Zulauf_RA_V.Stoerung.Res_23 := FALSE;
   Zulauf_RA_V.Stoerung.Res_24 := FALSE;
   Zulauf_RA_V.Stoerung.Res_25 := FALSE;
   Zulauf_RA_V.Stoerung.Res_26 := FALSE;
   Zulauf_RA_V.Stoerung.Res_27 := FALSE;
   Zulauf_RA_V.Stoerung.Res_28 := FALSE;
   Zulauf_RA_V.Stoerung.Res_29 := FALSE;
   Zulauf_RA_V.Stoerung.Res_30 := FALSE;
   Zulauf_RA_V.Stoerung.Res_31 := FALSE;
   Zulauf_RA_V.MW_I := 0.0;
   Zulauf_RA_V.MW_P := 0.0;
   Zulauf_RA_V.EZ := 0;
   Zulauf_RA_V.BZ_akt := 453021;
   Zulauf_RA_V.BZ_ges := 968974;
   Zulauf_RA_V.AZ_akt := 0;
   Zulauf_RA_V.ESH := 2;
   Zulauf_RA_V.SW_akt := 0.0;
   Zulauf_RA_V.SW_Auto := 0.0;
   Zulauf_RA_V.SW_out := 0.0;
   Zulauf_RA_RP.Status.Bed_vOrt := FALSE;
   Zulauf_RA_RP.Status.Bed_UV := FALSE;
   Zulauf_RA_RP.Status.Bed_NHV := TRUE;
   Zulauf_RA_RP.Status.Bed_PLS := FALSE;
   Zulauf_RA_RP.Status.BA_Hand := FALSE;
   Zulauf_RA_RP.Status.BA_Auto := TRUE;
   Zulauf_RA_RP.Status.RB_Ein1 := FALSE;
   Zulauf_RA_RP.Status.RB_Ein2 := FALSE;
   Zulauf_RA_RP.Status.RB_Aus := TRUE;
   Zulauf_RA_RP.Status.BFR_NS := FALSE;
   Zulauf_RA_RP.Status.BFR_ECS := FALSE;
   Zulauf_RA_RP.Status.BFR_ESK := FALSE;
   Zulauf_RA_RP.Status.BFR_MAZ := FALSE;
   Zulauf_RA_RP.Status.BFR_Rev := FALSE;
   Zulauf_RA_RP.Status.BFR_Ein1 := FALSE;
   Zulauf_RA_RP.Status.BFR_Ein2 := FALSE;
   Zulauf_RA_RP.Status.BM_Ein1 := FALSE;
   Zulauf_RA_RP.Status.BM_Ein2 := FALSE;
   Zulauf_RA_RP.Status.BM_Auf := FALSE;
   Zulauf_RA_RP.Status.BM_Zu := FALSE;
   Zulauf_RA_RP.Status.BM_Ein := FALSE;
   Zulauf_RA_RP.Status.BM_Aus := TRUE;
   Zulauf_RA_RP.Status.BM_Anst1 := FALSE;
   Zulauf_RA_RP.Status.BM_Anst2 := FALSE;
   Zulauf_RA_RP.Status.BM_Auto1 := FALSE;
   Zulauf_RA_RP.Status.BM_Auto2 := FALSE;
   Zulauf_RA_RP.Status.Res_26 := FALSE;
   Zulauf_RA_RP.Status.Res_27 := FALSE;
   Zulauf_RA_RP.Status.BB_NA := FALSE;
   Zulauf_RA_RP.Status.BB_AutoOk := TRUE;
   Zulauf_RA_RP.Status.BB_SS := FALSE;
   Zulauf_RA_RP.Status.BB_SSnq := FALSE;
   Zulauf_RA_RP.Stoerung.St_allg := FALSE;
   Zulauf_RA_RP.Stoerung.St_DMA := FALSE;
   Zulauf_RA_RP.Stoerung.St_DMZ := FALSE;
   Zulauf_RA_RP.Stoerung.St_FU := FALSE;
   Zulauf_RA_RP.Stoerung.St_TL := FALSE;
   Zulauf_RA_RP.Stoerung.St_UDr := FALSE;
   Zulauf_RA_RP.Stoerung.St_UeDr := FALSE;
   Zulauf_RA_RP.Stoerung.St_UeTemp := FALSE;
   Zulauf_RA_RP.Stoerung.St_Leck := FALSE;
   Zulauf_RA_RP.Stoerung.St_UeLM := FALSE;
   Zulauf_RA_RP.Stoerung.St_UeLE := FALSE;
   Zulauf_RA_RP.Stoerung.St_Kom_DP := FALSE;
   Zulauf_RA_RP.Stoerung.St_Kom_int := FALSE;
   Zulauf_RA_RP.Stoerung.St_int := FALSE;
   Zulauf_RA_RP.Stoerung.St_LZ := FALSE;
   Zulauf_RA_RP.Stoerung.St_BefLZ := FALSE;
   Zulauf_RA_RP.Stoerung.Wa_EZ := FALSE;
   Zulauf_RA_RP.Stoerung.Wa_Wart := FALSE;
   Zulauf_RA_RP.Stoerung.St_Strm := FALSE;
   Zulauf_RA_RP.Stoerung.Res_19 := FALSE;
   Zulauf_RA_RP.Stoerung.Res_20 := FALSE;
   Zulauf_RA_RP.Stoerung.Res_21 := FALSE;
   Zulauf_RA_RP.Stoerung.Res_22 := FALSE;
   Zulauf_RA_RP.Stoerung.Res_23 := FALSE;
   Zulauf_RA_RP.Stoerung.Res_24 := FALSE;
   Zulauf_RA_RP.Stoerung.Res_25 := FALSE;
   Zulauf_RA_RP.Stoerung.Res_26 := FALSE;
   Zulauf_RA_RP.Stoerung.Res_27 := FALSE;
   Zulauf_RA_RP.Stoerung.Res_28 := FALSE;
   Zulauf_RA_RP.Stoerung.Res_29 := FALSE;
   Zulauf_RA_RP.Stoerung.Res_30 := FALSE;
   Zulauf_RA_RP.Stoerung.Res_31 := FALSE;
   Zulauf_RA_RP.MW_I := 0.0;
   Zulauf_RA_RP.MW_P := 0.0;
   Zulauf_RA_RP.EZ := 0;
   Zulauf_RA_RP.BZ_akt := 4;
   Zulauf_RA_RP.BZ_ges := 714;
   Zulauf_RA_RP.AZ_akt := 191744;
   Zulauf_RA_RP.ESH := 32;
   Zulauf_RA_RP.SW_akt := 0.0;
   Zulauf_RA_RP.SW_Auto := 0.0;
   Zulauf_RA_RP.SW_out := 0.0;
   Zulauf_RA_FP.Status.Bed_vOrt := FALSE;
   Zulauf_RA_FP.Status.Bed_UV := FALSE;
   Zulauf_RA_FP.Status.Bed_NHV := TRUE;
   Zulauf_RA_FP.Status.Bed_PLS := FALSE;
   Zulauf_RA_FP.Status.BA_Hand := FALSE;
   Zulauf_RA_FP.Status.BA_Auto := TRUE;
   Zulauf_RA_FP.Status.RB_Ein1 := FALSE;
   Zulauf_RA_FP.Status.RB_Ein2 := FALSE;
   Zulauf_RA_FP.Status.RB_Aus := TRUE;
   Zulauf_RA_FP.Status.BFR_NS := FALSE;
   Zulauf_RA_FP.Status.BFR_ECS := FALSE;
   Zulauf_RA_FP.Status.BFR_ESK := FALSE;
   Zulauf_RA_FP.Status.BFR_MAZ := FALSE;
   Zulauf_RA_FP.Status.BFR_Rev := FALSE;
   Zulauf_RA_FP.Status.BFR_Ein1 := FALSE;
   Zulauf_RA_FP.Status.BFR_Ein2 := FALSE;
   Zulauf_RA_FP.Status.BM_Ein1 := FALSE;
   Zulauf_RA_FP.Status.BM_Ein2 := FALSE;
   Zulauf_RA_FP.Status.BM_Auf := FALSE;
   Zulauf_RA_FP.Status.BM_Zu := FALSE;
   Zulauf_RA_FP.Status.BM_Ein := FALSE;
   Zulauf_RA_FP.Status.BM_Aus := TRUE;
   Zulauf_RA_FP.Status.BM_Anst1 := FALSE;
   Zulauf_RA_FP.Status.BM_Anst2 := FALSE;
   Zulauf_RA_FP.Status.BM_Auto1 := FALSE;
   Zulauf_RA_FP.Status.BM_Auto2 := FALSE;
   Zulauf_RA_FP.Status.Res_26 := FALSE;
   Zulauf_RA_FP.Status.Res_27 := FALSE;
   Zulauf_RA_FP.Status.BB_NA := FALSE;
   Zulauf_RA_FP.Status.BB_AutoOk := TRUE;
   Zulauf_RA_FP.Status.BB_SS := FALSE;
   Zulauf_RA_FP.Status.BB_SSnq := FALSE;
   Zulauf_RA_FP.Stoerung.St_allg := FALSE;
   Zulauf_RA_FP.Stoerung.St_DMA := FALSE;
   Zulauf_RA_FP.Stoerung.St_DMZ := FALSE;
   Zulauf_RA_FP.Stoerung.St_FU := FALSE;
   Zulauf_RA_FP.Stoerung.St_TL := FALSE;
   Zulauf_RA_FP.Stoerung.St_UDr := FALSE;
   Zulauf_RA_FP.Stoerung.St_UeDr := FALSE;
   Zulauf_RA_FP.Stoerung.St_UeTemp := FALSE;
   Zulauf_RA_FP.Stoerung.St_Leck := FALSE;
   Zulauf_RA_FP.Stoerung.St_UeLM := FALSE;
   Zulauf_RA_FP.Stoerung.St_UeLE := FALSE;
   Zulauf_RA_FP.Stoerung.St_Kom_DP := FALSE;
   Zulauf_RA_FP.Stoerung.St_Kom_int := FALSE;
   Zulauf_RA_FP.Stoerung.St_int := FALSE;
   Zulauf_RA_FP.Stoerung.St_LZ := FALSE;
   Zulauf_RA_FP.Stoerung.St_BefLZ := FALSE;
   Zulauf_RA_FP.Stoerung.Wa_EZ := FALSE;
   Zulauf_RA_FP.Stoerung.Wa_Wart := FALSE;
   Zulauf_RA_FP.Stoerung.St_Strm := FALSE;
   Zulauf_RA_FP.Stoerung.Res_19 := FALSE;
   Zulauf_RA_FP.Stoerung.Res_20 := FALSE;
   Zulauf_RA_FP.Stoerung.Res_21 := FALSE;
   Zulauf_RA_FP.Stoerung.Res_22 := FALSE;
   Zulauf_RA_FP.Stoerung.Res_23 := FALSE;
   Zulauf_RA_FP.Stoerung.Res_24 := FALSE;
   Zulauf_RA_FP.Stoerung.Res_25 := FALSE;
   Zulauf_RA_FP.Stoerung.Res_26 := FALSE;
   Zulauf_RA_FP.Stoerung.Res_27 := FALSE;
   Zulauf_RA_FP.Stoerung.Res_28 := FALSE;
   Zulauf_RA_FP.Stoerung.Res_29 := FALSE;
   Zulauf_RA_FP.Stoerung.Res_30 := FALSE;
   Zulauf_RA_FP.Stoerung.Res_31 := FALSE;
   Zulauf_RA_FP.MW_I := 0.0;
   Zulauf_RA_FP.MW_P := 0.0;
   Zulauf_RA_FP.EZ := 0;
   Zulauf_RA_FP.BZ_akt := 63;
   Zulauf_RA_FP.BZ_ges := 629;
   Zulauf_RA_FP.AZ_akt := 191748;
   Zulauf_RA_FP.ESH := 9;
   Zulauf_RA_FP.SW_akt := 0.0;
   Zulauf_RA_FP.SW_Auto := 0.0;
   Zulauf_RA_FP.SW_out := 0.0;
   Schlamm_BP.Status.Bed_vOrt := FALSE;
   Schlamm_BP.Status.Bed_UV := FALSE;
   Schlamm_BP.Status.Bed_NHV := FALSE;
   Schlamm_BP.Status.Bed_PLS := TRUE;
   Schlamm_BP.Status.BA_Hand := FALSE;
   Schlamm_BP.Status.BA_Auto := TRUE;
   Schlamm_BP.Status.RB_Ein1 := FALSE;
   Schlamm_BP.Status.RB_Ein2 := FALSE;
   Schlamm_BP.Status.RB_Aus := TRUE;
   Schlamm_BP.Status.BFR_NS := FALSE;
   Schlamm_BP.Status.BFR_ECS := FALSE;
   Schlamm_BP.Status.BFR_ESK := FALSE;
   Schlamm_BP.Status.BFR_MAZ := FALSE;
   Schlamm_BP.Status.BFR_Rev := FALSE;
   Schlamm_BP.Status.BFR_Ein1 := FALSE;
   Schlamm_BP.Status.BFR_Ein2 := FALSE;
   Schlamm_BP.Status.BM_Ein1 := FALSE;
   Schlamm_BP.Status.BM_Ein2 := FALSE;
   Schlamm_BP.Status.BM_Auf := FALSE;
   Schlamm_BP.Status.BM_Zu := FALSE;
   Schlamm_BP.Status.BM_Ein := FALSE;
   Schlamm_BP.Status.BM_Aus := TRUE;
   Schlamm_BP.Status.BM_Anst1 := FALSE;
   Schlamm_BP.Status.BM_Anst2 := FALSE;
   Schlamm_BP.Status.BM_Auto1 := FALSE;
   Schlamm_BP.Status.BM_Auto2 := FALSE;
   Schlamm_BP.Status.Res_26 := FALSE;
   Schlamm_BP.Status.Res_27 := FALSE;
   Schlamm_BP.Status.BB_NA := FALSE;
   Schlamm_BP.Status.BB_AutoOk := TRUE;
   Schlamm_BP.Status.BB_SS := FALSE;
   Schlamm_BP.Status.BB_SSnq := FALSE;
   Schlamm_BP.Stoerung.St_allg := FALSE;
   Schlamm_BP.Stoerung.St_DMA := FALSE;
   Schlamm_BP.Stoerung.St_DMZ := FALSE;
   Schlamm_BP.Stoerung.St_FU := FALSE;
   Schlamm_BP.Stoerung.St_TL := FALSE;
   Schlamm_BP.Stoerung.St_UDr := FALSE;
   Schlamm_BP.Stoerung.St_UeDr := FALSE;
   Schlamm_BP.Stoerung.St_UeTemp := FALSE;
   Schlamm_BP.Stoerung.St_Leck := FALSE;
   Schlamm_BP.Stoerung.St_UeLM := FALSE;
   Schlamm_BP.Stoerung.St_UeLE := FALSE;
   Schlamm_BP.Stoerung.St_Kom_DP := FALSE;
   Schlamm_BP.Stoerung.St_Kom_int := FALSE;
   Schlamm_BP.Stoerung.St_int := FALSE;
   Schlamm_BP.Stoerung.St_LZ := FALSE;
   Schlamm_BP.Stoerung.St_BefLZ := FALSE;
   Schlamm_BP.Stoerung.Wa_EZ := FALSE;
   Schlamm_BP.Stoerung.Wa_Wart := FALSE;
   Schlamm_BP.Stoerung.St_Strm := FALSE;
   Schlamm_BP.Stoerung.Res_19 := FALSE;
   Schlamm_BP.Stoerung.Res_20 := FALSE;
   Schlamm_BP.Stoerung.Res_21 := FALSE;
   Schlamm_BP.Stoerung.Res_22 := FALSE;
   Schlamm_BP.Stoerung.Res_23 := FALSE;
   Schlamm_BP.Stoerung.Res_24 := FALSE;
   Schlamm_BP.Stoerung.Res_25 := FALSE;
   Schlamm_BP.Stoerung.Res_26 := FALSE;
   Schlamm_BP.Stoerung.Res_27 := FALSE;
   Schlamm_BP.Stoerung.Res_28 := FALSE;
   Schlamm_BP.Stoerung.Res_29 := FALSE;
   Schlamm_BP.Stoerung.Res_30 := FALSE;
   Schlamm_BP.Stoerung.Res_31 := FALSE;
   Schlamm_BP.MW_I := 0.0;
   Schlamm_BP.MW_P := 0.0;
   Schlamm_BP.EZ := 0;
   Schlamm_BP.BZ_akt := 2540;
   Schlamm_BP.BZ_ges := 2744811;
   Schlamm_BP.AZ_akt := 14567;
   Schlamm_BP.ESH := 1061;
   Schlamm_BP.SW_akt := 0.0;
   Schlamm_BP.SW_Auto := 0.0;
   Schlamm_BP.SW_out := 0.0;
   Truebwasser_P1.Status.Bed_vOrt := FALSE;
   Truebwasser_P1.Status.Bed_UV := FALSE;
   Truebwasser_P1.Status.Bed_NHV := FALSE;
   Truebwasser_P1.Status.Bed_PLS := TRUE;
   Truebwasser_P1.Status.BA_Hand := FALSE;
   Truebwasser_P1.Status.BA_Auto := TRUE;
   Truebwasser_P1.Status.RB_Ein1 := FALSE;
   Truebwasser_P1.Status.RB_Ein2 := FALSE;
   Truebwasser_P1.Status.RB_Aus := TRUE;
   Truebwasser_P1.Status.BFR_NS := FALSE;
   Truebwasser_P1.Status.BFR_ECS := FALSE;
   Truebwasser_P1.Status.BFR_ESK := FALSE;
   Truebwasser_P1.Status.BFR_MAZ := FALSE;
   Truebwasser_P1.Status.BFR_Rev := FALSE;
   Truebwasser_P1.Status.BFR_Ein1 := FALSE;
   Truebwasser_P1.Status.BFR_Ein2 := FALSE;
   Truebwasser_P1.Status.BM_Ein1 := FALSE;
   Truebwasser_P1.Status.BM_Ein2 := FALSE;
   Truebwasser_P1.Status.BM_Auf := FALSE;
   Truebwasser_P1.Status.BM_Zu := FALSE;
   Truebwasser_P1.Status.BM_Ein := FALSE;
   Truebwasser_P1.Status.BM_Aus := TRUE;
   Truebwasser_P1.Status.BM_Anst1 := FALSE;
   Truebwasser_P1.Status.BM_Anst2 := FALSE;
   Truebwasser_P1.Status.BM_Auto1 := FALSE;
   Truebwasser_P1.Status.BM_Auto2 := FALSE;
   Truebwasser_P1.Status.Res_26 := FALSE;
   Truebwasser_P1.Status.Res_27 := FALSE;
   Truebwasser_P1.Status.BB_NA := FALSE;
   Truebwasser_P1.Status.BB_AutoOk := TRUE;
   Truebwasser_P1.Status.BB_SS := FALSE;
   Truebwasser_P1.Status.BB_SSnq := FALSE;
   Truebwasser_P1.Stoerung.St_allg := FALSE;
   Truebwasser_P1.Stoerung.St_DMA := FALSE;
   Truebwasser_P1.Stoerung.St_DMZ := FALSE;
   Truebwasser_P1.Stoerung.St_FU := FALSE;
   Truebwasser_P1.Stoerung.St_TL := FALSE;
   Truebwasser_P1.Stoerung.St_UDr := FALSE;
   Truebwasser_P1.Stoerung.St_UeDr := FALSE;
   Truebwasser_P1.Stoerung.St_UeTemp := FALSE;
   Truebwasser_P1.Stoerung.St_Leck := FALSE;
   Truebwasser_P1.Stoerung.St_UeLM := FALSE;
   Truebwasser_P1.Stoerung.St_UeLE := FALSE;
   Truebwasser_P1.Stoerung.St_Kom_DP := FALSE;
   Truebwasser_P1.Stoerung.St_Kom_int := FALSE;
   Truebwasser_P1.Stoerung.St_int := FALSE;
   Truebwasser_P1.Stoerung.St_LZ := FALSE;
   Truebwasser_P1.Stoerung.St_BefLZ := FALSE;
   Truebwasser_P1.Stoerung.Wa_EZ := FALSE;
   Truebwasser_P1.Stoerung.Wa_Wart := FALSE;
   Truebwasser_P1.Stoerung.St_Strm := FALSE;
   Truebwasser_P1.Stoerung.Res_19 := FALSE;
   Truebwasser_P1.Stoerung.Res_20 := FALSE;
   Truebwasser_P1.Stoerung.Res_21 := FALSE;
   Truebwasser_P1.Stoerung.Res_22 := FALSE;
   Truebwasser_P1.Stoerung.Res_23 := FALSE;
   Truebwasser_P1.Stoerung.Res_24 := FALSE;
   Truebwasser_P1.Stoerung.Res_25 := FALSE;
   Truebwasser_P1.Stoerung.Res_26 := FALSE;
   Truebwasser_P1.Stoerung.Res_27 := FALSE;
   Truebwasser_P1.Stoerung.Res_28 := FALSE;
   Truebwasser_P1.Stoerung.Res_29 := FALSE;
   Truebwasser_P1.Stoerung.Res_30 := FALSE;
   Truebwasser_P1.Stoerung.Res_31 := FALSE;
   Truebwasser_P1.MW_I := 0.0;
   Truebwasser_P1.MW_P := 0.0;
   Truebwasser_P1.EZ := 0;
   Truebwasser_P1.BZ_akt := 8026;
   Truebwasser_P1.BZ_ges := 27425188;
   Truebwasser_P1.AZ_akt := 440685;
   Truebwasser_P1.ESH := 4849;
   Truebwasser_P1.SW_akt := 0.0;
   Truebwasser_P1.SW_Auto := 0.0;
   Truebwasser_P1.SW_out := 0.0;
   Truebwasser_P2.Status.Bed_vOrt := FALSE;
   Truebwasser_P2.Status.Bed_UV := FALSE;
   Truebwasser_P2.Status.Bed_NHV := FALSE;
   Truebwasser_P2.Status.Bed_PLS := TRUE;
   Truebwasser_P2.Status.BA_Hand := FALSE;
   Truebwasser_P2.Status.BA_Auto := TRUE;
   Truebwasser_P2.Status.RB_Ein1 := FALSE;
   Truebwasser_P2.Status.RB_Ein2 := FALSE;
   Truebwasser_P2.Status.RB_Aus := TRUE;
   Truebwasser_P2.Status.BFR_NS := FALSE;
   Truebwasser_P2.Status.BFR_ECS := FALSE;
   Truebwasser_P2.Status.BFR_ESK := FALSE;
   Truebwasser_P2.Status.BFR_MAZ := FALSE;
   Truebwasser_P2.Status.BFR_Rev := FALSE;
   Truebwasser_P2.Status.BFR_Ein1 := FALSE;
   Truebwasser_P2.Status.BFR_Ein2 := FALSE;
   Truebwasser_P2.Status.BM_Ein1 := FALSE;
   Truebwasser_P2.Status.BM_Ein2 := FALSE;
   Truebwasser_P2.Status.BM_Auf := FALSE;
   Truebwasser_P2.Status.BM_Zu := FALSE;
   Truebwasser_P2.Status.BM_Ein := FALSE;
   Truebwasser_P2.Status.BM_Aus := TRUE;
   Truebwasser_P2.Status.BM_Anst1 := FALSE;
   Truebwasser_P2.Status.BM_Anst2 := FALSE;
   Truebwasser_P2.Status.BM_Auto1 := FALSE;
   Truebwasser_P2.Status.BM_Auto2 := FALSE;
   Truebwasser_P2.Status.Res_26 := FALSE;
   Truebwasser_P2.Status.Res_27 := FALSE;
   Truebwasser_P2.Status.BB_NA := FALSE;
   Truebwasser_P2.Status.BB_AutoOk := TRUE;
   Truebwasser_P2.Status.BB_SS := FALSE;
   Truebwasser_P2.Status.BB_SSnq := FALSE;
   Truebwasser_P2.Stoerung.St_allg := FALSE;
   Truebwasser_P2.Stoerung.St_DMA := FALSE;
   Truebwasser_P2.Stoerung.St_DMZ := FALSE;
   Truebwasser_P2.Stoerung.St_FU := FALSE;
   Truebwasser_P2.Stoerung.St_TL := FALSE;
   Truebwasser_P2.Stoerung.St_UDr := FALSE;
   Truebwasser_P2.Stoerung.St_UeDr := FALSE;
   Truebwasser_P2.Stoerung.St_UeTemp := FALSE;
   Truebwasser_P2.Stoerung.St_Leck := FALSE;
   Truebwasser_P2.Stoerung.St_UeLM := FALSE;
   Truebwasser_P2.Stoerung.St_UeLE := FALSE;
   Truebwasser_P2.Stoerung.St_Kom_DP := FALSE;
   Truebwasser_P2.Stoerung.St_Kom_int := FALSE;
   Truebwasser_P2.Stoerung.St_int := FALSE;
   Truebwasser_P2.Stoerung.St_LZ := FALSE;
   Truebwasser_P2.Stoerung.St_BefLZ := FALSE;
   Truebwasser_P2.Stoerung.Wa_EZ := FALSE;
   Truebwasser_P2.Stoerung.Wa_Wart := FALSE;
   Truebwasser_P2.Stoerung.St_Strm := FALSE;
   Truebwasser_P2.Stoerung.Res_19 := FALSE;
   Truebwasser_P2.Stoerung.Res_20 := FALSE;
   Truebwasser_P2.Stoerung.Res_21 := FALSE;
   Truebwasser_P2.Stoerung.Res_22 := FALSE;
   Truebwasser_P2.Stoerung.Res_23 := FALSE;
   Truebwasser_P2.Stoerung.Res_24 := FALSE;
   Truebwasser_P2.Stoerung.Res_25 := FALSE;
   Truebwasser_P2.Stoerung.Res_26 := FALSE;
   Truebwasser_P2.Stoerung.Res_27 := FALSE;
   Truebwasser_P2.Stoerung.Res_28 := FALSE;
   Truebwasser_P2.Stoerung.Res_29 := FALSE;
   Truebwasser_P2.Stoerung.Res_30 := FALSE;
   Truebwasser_P2.Stoerung.Res_31 := FALSE;
   Truebwasser_P2.MW_I := 0.0;
   Truebwasser_P2.MW_P := 0.0;
   Truebwasser_P2.EZ := 0;
   Truebwasser_P2.BZ_akt := 8061;
   Truebwasser_P2.BZ_ges := 22596981;
   Truebwasser_P2.AZ_akt := 34582;
   Truebwasser_P2.ESH := 4252;
   Truebwasser_P2.SW_akt := 0.0;
   Truebwasser_P2.SW_Auto := 0.0;
   Truebwasser_P2.SW_out := 0.0;
   Schlamm_AS.Status.Bed_vOrt := FALSE;
   Schlamm_AS.Status.Bed_UV := FALSE;
   Schlamm_AS.Status.Bed_NHV := FALSE;
   Schlamm_AS.Status.Bed_PLS := TRUE;
   Schlamm_AS.Status.BA_Hand := FALSE;
   Schlamm_AS.Status.BA_Auto := TRUE;
   Schlamm_AS.Status.RB_Ein1 := FALSE;
   Schlamm_AS.Status.RB_Ein2 := FALSE;
   Schlamm_AS.Status.RB_Aus := TRUE;
   Schlamm_AS.Status.BFR_NS := FALSE;
   Schlamm_AS.Status.BFR_ECS := FALSE;
   Schlamm_AS.Status.BFR_ESK := FALSE;
   Schlamm_AS.Status.BFR_MAZ := FALSE;
   Schlamm_AS.Status.BFR_Rev := FALSE;
   Schlamm_AS.Status.BFR_Ein1 := FALSE;
   Schlamm_AS.Status.BFR_Ein2 := FALSE;
   Schlamm_AS.Status.BM_Ein1 := FALSE;
   Schlamm_AS.Status.BM_Ein2 := FALSE;
   Schlamm_AS.Status.BM_Auf := FALSE;
   Schlamm_AS.Status.BM_Zu := TRUE;
   Schlamm_AS.Status.BM_Ein := FALSE;
   Schlamm_AS.Status.BM_Aus := TRUE;
   Schlamm_AS.Status.BM_Anst1 := FALSE;
   Schlamm_AS.Status.BM_Anst2 := FALSE;
   Schlamm_AS.Status.BM_Auto1 := FALSE;
   Schlamm_AS.Status.BM_Auto2 := TRUE;
   Schlamm_AS.Status.Res_26 := FALSE;
   Schlamm_AS.Status.Res_27 := FALSE;
   Schlamm_AS.Status.BB_NA := FALSE;
   Schlamm_AS.Status.BB_AutoOk := TRUE;
   Schlamm_AS.Status.BB_SS := FALSE;
   Schlamm_AS.Status.BB_SSnq := FALSE;
   Schlamm_AS.Stoerung.St_allg := FALSE;
   Schlamm_AS.Stoerung.St_DMA := FALSE;
   Schlamm_AS.Stoerung.St_DMZ := FALSE;
   Schlamm_AS.Stoerung.St_FU := FALSE;
   Schlamm_AS.Stoerung.St_TL := FALSE;
   Schlamm_AS.Stoerung.St_UDr := FALSE;
   Schlamm_AS.Stoerung.St_UeDr := FALSE;
   Schlamm_AS.Stoerung.St_UeTemp := FALSE;
   Schlamm_AS.Stoerung.St_Leck := FALSE;
   Schlamm_AS.Stoerung.St_UeLM := FALSE;
   Schlamm_AS.Stoerung.St_UeLE := FALSE;
   Schlamm_AS.Stoerung.St_Kom_DP := FALSE;
   Schlamm_AS.Stoerung.St_Kom_int := FALSE;
   Schlamm_AS.Stoerung.St_int := FALSE;
   Schlamm_AS.Stoerung.St_LZ := FALSE;
   Schlamm_AS.Stoerung.St_BefLZ := FALSE;
   Schlamm_AS.Stoerung.Wa_EZ := FALSE;
   Schlamm_AS.Stoerung.Wa_Wart := FALSE;
   Schlamm_AS.Stoerung.St_Strm := FALSE;
   Schlamm_AS.Stoerung.Res_19 := FALSE;
   Schlamm_AS.Stoerung.Res_20 := FALSE;
   Schlamm_AS.Stoerung.Res_21 := FALSE;
   Schlamm_AS.Stoerung.Res_22 := FALSE;
   Schlamm_AS.Stoerung.Res_23 := FALSE;
   Schlamm_AS.Stoerung.Res_24 := FALSE;
   Schlamm_AS.Stoerung.Res_25 := FALSE;
   Schlamm_AS.Stoerung.Res_26 := FALSE;
   Schlamm_AS.Stoerung.Res_27 := FALSE;
   Schlamm_AS.Stoerung.Res_28 := FALSE;
   Schlamm_AS.Stoerung.Res_29 := FALSE;
   Schlamm_AS.Stoerung.Res_30 := FALSE;
   Schlamm_AS.Stoerung.Res_31 := FALSE;
   Schlamm_AS.MW_I := 0.0;
   Schlamm_AS.MW_P := 0.0;
   Schlamm_AS.EZ := 0;
   Schlamm_AS.BZ_akt := 34;
   Schlamm_AS.BZ_ges := 70689;
   Schlamm_AS.AZ_akt := 14533;
   Schlamm_AS.ESH := 2093;
   Schlamm_AS.SW_akt := 0.0;
   Schlamm_AS.SW_Auto := 0.0;
   Schlamm_AS.SW_out := 0.0;
   BB2_SR_K.Status.Bed_vOrt := FALSE;
   BB2_SR_K.Status.Bed_UV := FALSE;
   BB2_SR_K.Status.Bed_NHV := TRUE;
   BB2_SR_K.Status.Bed_PLS := FALSE;
   BB2_SR_K.Status.BA_Hand := FALSE;
   BB2_SR_K.Status.BA_Auto := TRUE;
   BB2_SR_K.Status.RB_Ein1 := FALSE;
   BB2_SR_K.Status.RB_Ein2 := FALSE;
   BB2_SR_K.Status.RB_Aus := TRUE;
   BB2_SR_K.Status.BFR_NS := FALSE;
   BB2_SR_K.Status.BFR_ECS := FALSE;
   BB2_SR_K.Status.BFR_ESK := FALSE;
   BB2_SR_K.Status.BFR_MAZ := FALSE;
   BB2_SR_K.Status.BFR_Rev := FALSE;
   BB2_SR_K.Status.BFR_Ein1 := FALSE;
   BB2_SR_K.Status.BFR_Ein2 := FALSE;
   BB2_SR_K.Status.BM_Ein1 := FALSE;
   BB2_SR_K.Status.BM_Ein2 := FALSE;
   BB2_SR_K.Status.BM_Auf := FALSE;
   BB2_SR_K.Status.BM_Zu := FALSE;
   BB2_SR_K.Status.BM_Ein := FALSE;
   BB2_SR_K.Status.BM_Aus := TRUE;
   BB2_SR_K.Status.BM_Anst1 := FALSE;
   BB2_SR_K.Status.BM_Anst2 := FALSE;
   BB2_SR_K.Status.BM_Auto1 := FALSE;
   BB2_SR_K.Status.BM_Auto2 := FALSE;
   BB2_SR_K.Status.Res_26 := FALSE;
   BB2_SR_K.Status.Res_27 := FALSE;
   BB2_SR_K.Status.BB_NA := FALSE;
   BB2_SR_K.Status.BB_AutoOk := TRUE;
   BB2_SR_K.Status.BB_SS := FALSE;
   BB2_SR_K.Status.BB_SSnq := FALSE;
   BB2_SR_K.Stoerung.St_allg := FALSE;
   BB2_SR_K.Stoerung.St_DMA := FALSE;
   BB2_SR_K.Stoerung.St_DMZ := FALSE;
   BB2_SR_K.Stoerung.St_FU := FALSE;
   BB2_SR_K.Stoerung.St_TL := FALSE;
   BB2_SR_K.Stoerung.St_UDr := FALSE;
   BB2_SR_K.Stoerung.St_UeDr := FALSE;
   BB2_SR_K.Stoerung.St_UeTemp := FALSE;
   BB2_SR_K.Stoerung.St_Leck := FALSE;
   BB2_SR_K.Stoerung.St_UeLM := FALSE;
   BB2_SR_K.Stoerung.St_UeLE := FALSE;
   BB2_SR_K.Stoerung.St_Kom_DP := FALSE;
   BB2_SR_K.Stoerung.St_Kom_int := FALSE;
   BB2_SR_K.Stoerung.St_int := FALSE;
   BB2_SR_K.Stoerung.St_LZ := FALSE;
   BB2_SR_K.Stoerung.St_BefLZ := FALSE;
   BB2_SR_K.Stoerung.Wa_EZ := FALSE;
   BB2_SR_K.Stoerung.Wa_Wart := FALSE;
   BB2_SR_K.Stoerung.St_Strm := FALSE;
   BB2_SR_K.Stoerung.Res_19 := FALSE;
   BB2_SR_K.Stoerung.Res_20 := FALSE;
   BB2_SR_K.Stoerung.Res_21 := FALSE;
   BB2_SR_K.Stoerung.Res_22 := FALSE;
   BB2_SR_K.Stoerung.Res_23 := FALSE;
   BB2_SR_K.Stoerung.Res_24 := FALSE;
   BB2_SR_K.Stoerung.Res_25 := FALSE;
   BB2_SR_K.Stoerung.Res_26 := FALSE;
   BB2_SR_K.Stoerung.Res_27 := FALSE;
   BB2_SR_K.Stoerung.Res_28 := FALSE;
   BB2_SR_K.Stoerung.Res_29 := FALSE;
   BB2_SR_K.Stoerung.Res_30 := FALSE;
   BB2_SR_K.Stoerung.Res_31 := FALSE;
   BB2_SR_K.MW_I := 0.0;
   BB2_SR_K.MW_P := 0.0;
   BB2_SR_K.EZ := 0;
   BB2_SR_K.BZ_akt := 179;
   BB2_SR_K.BZ_ges := 6115705;
   BB2_SR_K.AZ_akt := 1985;
   BB2_SR_K.ESH := 34083;
   BB2_SR_K.SW_akt := 0.0;
   BB2_SR_K.SW_Auto := 0.0;
   BB2_SR_K.SW_out := 0.0;
   Zulauf_DosP.Status.Bed_vOrt := FALSE;
   Zulauf_DosP.Status.Bed_UV := FALSE;
   Zulauf_DosP.Status.Bed_NHV := FALSE;
   Zulauf_DosP.Status.Bed_PLS := TRUE;
   Zulauf_DosP.Status.BA_Hand := FALSE;
   Zulauf_DosP.Status.BA_Auto := TRUE;
   Zulauf_DosP.Status.RB_Ein1 := TRUE;
   Zulauf_DosP.Status.RB_Ein2 := FALSE;
   Zulauf_DosP.Status.RB_Aus := FALSE;
   Zulauf_DosP.Status.BFR_NS := FALSE;
   Zulauf_DosP.Status.BFR_ECS := FALSE;
   Zulauf_DosP.Status.BFR_ESK := FALSE;
   Zulauf_DosP.Status.BFR_MAZ := FALSE;
   Zulauf_DosP.Status.BFR_Rev := FALSE;
   Zulauf_DosP.Status.BFR_Ein1 := FALSE;
   Zulauf_DosP.Status.BFR_Ein2 := FALSE;
   Zulauf_DosP.Status.BM_Ein1 := TRUE;
   Zulauf_DosP.Status.BM_Ein2 := FALSE;
   Zulauf_DosP.Status.BM_Auf := FALSE;
   Zulauf_DosP.Status.BM_Zu := FALSE;
   Zulauf_DosP.Status.BM_Ein := TRUE;
   Zulauf_DosP.Status.BM_Aus := FALSE;
   Zulauf_DosP.Status.BM_Anst1 := TRUE;
   Zulauf_DosP.Status.BM_Anst2 := FALSE;
   Zulauf_DosP.Status.BM_Auto1 := TRUE;
   Zulauf_DosP.Status.BM_Auto2 := FALSE;
   Zulauf_DosP.Status.Res_26 := FALSE;
   Zulauf_DosP.Status.Res_27 := FALSE;
   Zulauf_DosP.Status.BB_NA := FALSE;
   Zulauf_DosP.Status.BB_AutoOk := TRUE;
   Zulauf_DosP.Status.BB_SS := FALSE;
   Zulauf_DosP.Status.BB_SSnq := FALSE;
   Zulauf_DosP.Stoerung.St_allg := FALSE;
   Zulauf_DosP.Stoerung.St_DMA := FALSE;
   Zulauf_DosP.Stoerung.St_DMZ := FALSE;
   Zulauf_DosP.Stoerung.St_FU := FALSE;
   Zulauf_DosP.Stoerung.St_TL := FALSE;
   Zulauf_DosP.Stoerung.St_UDr := FALSE;
   Zulauf_DosP.Stoerung.St_UeDr := FALSE;
   Zulauf_DosP.Stoerung.St_UeTemp := FALSE;
   Zulauf_DosP.Stoerung.St_Leck := FALSE;
   Zulauf_DosP.Stoerung.St_UeLM := FALSE;
   Zulauf_DosP.Stoerung.St_UeLE := FALSE;
   Zulauf_DosP.Stoerung.St_Kom_DP := FALSE;
   Zulauf_DosP.Stoerung.St_Kom_int := FALSE;
   Zulauf_DosP.Stoerung.St_int := FALSE;
   Zulauf_DosP.Stoerung.St_LZ := FALSE;
   Zulauf_DosP.Stoerung.St_BefLZ := FALSE;
   Zulauf_DosP.Stoerung.Wa_EZ := FALSE;
   Zulauf_DosP.Stoerung.Wa_Wart := FALSE;
   Zulauf_DosP.Stoerung.St_Strm := FALSE;
   Zulauf_DosP.Stoerung.Res_19 := FALSE;
   Zulauf_DosP.Stoerung.Res_20 := FALSE;
   Zulauf_DosP.Stoerung.Res_21 := FALSE;
   Zulauf_DosP.Stoerung.Res_22 := FALSE;
   Zulauf_DosP.Stoerung.Res_23 := FALSE;
   Zulauf_DosP.Stoerung.Res_24 := FALSE;
   Zulauf_DosP.Stoerung.Res_25 := FALSE;
   Zulauf_DosP.Stoerung.Res_26 := FALSE;
   Zulauf_DosP.Stoerung.Res_27 := FALSE;
   Zulauf_DosP.Stoerung.Res_28 := FALSE;
   Zulauf_DosP.Stoerung.Res_29 := FALSE;
   Zulauf_DosP.Stoerung.Res_30 := FALSE;
   Zulauf_DosP.Stoerung.Res_31 := FALSE;
   Zulauf_DosP.MW_I := 0.0;
   Zulauf_DosP.MW_P := 0.0;
   Zulauf_DosP.EZ := 0;
   Zulauf_DosP.BZ_akt := 4714;
   Zulauf_DosP.BZ_ges := 40974809;
   Zulauf_DosP.AZ_akt := 224;
   Zulauf_DosP.ESH := 98;
   Zulauf_DosP.SW_akt := 0.3738;
   Zulauf_DosP.SW_Auto := 0.378229;
   Zulauf_DosP.SW_out := 0.378229;

END_DATA_BLOCK

DATA_BLOCK "DB106_Antriebe_Prm"
{ S7_Optimized_Access := 'FALSE' }
VERSION : 0.1
   STRUCT
      BB_G1 : "T_ANTRIEB_PRM";   // Belebung - Gebläse 1
      BB_G2 : "T_ANTRIEB_PRM";   // Belebung - Gebläse 2
      BB_G3 : "T_ANTRIEB_PRM";   // Belebung - Gebläse 3
      BB_SHL_G1 : "T_ANTRIEB_PRM";   // Belebung - Schallhaubenlüfter Gebläse 1
      BB_SHL_G2 : "T_ANTRIEB_PRM";   // Belebung - Schallhaubenlüfter Gebläse 2
      BB_SHL_G3 : "T_ANTRIEB_PRM";   // Belebung - Schallhaubenlüfter Gebläse 3
      BB_AV : "T_ANTRIEB_PRM";   // Belebung - Gebläsestation - Abluftventilator
      BB_LS1 : "T_ANTRIEB_PRM";   // Belebung - Gebläsestation - Luftwegschieber 1
      BB_LS2 : "T_ANTRIEB_PRM";   // Belebung - Gebläsestation - Luftwegschieber 2
      BB1_RZP1 : "T_ANTRIEB_PRM";   // Becken 1 - Rezipumpe 1
      BB1_RZP2 : "T_ANTRIEB_PRM";   // Becken 1 - Rezipumpe 2
      BB1_UeSP : "T_ANTRIEB_PRM";   // Becken 1 - ÜSS-Pumpe
      BB1_AS1 : "T_ANTRIEB_PRM";   // Becken 1 - Ablaufschieber 1
      BB1_AS2 : "T_ANTRIEB_PRM";   // Becken 1 - Ablaufschieber 2
      BB1_SR1 : "T_ANTRIEB_PRM";   // Becken 1 - MV Schlammrückführung 1
      BB1_SR2 : "T_ANTRIEB_PRM";   // Becken 1 - MV Schlammrückführung 2
      BB2_RZP1 : "T_ANTRIEB_PRM";   // Becken 2 - Rezipumpe 1
      BB2_RZP2 : "T_ANTRIEB_PRM";   // Becken 2 - Rezipumpe 2
      BB2_UeSP : "T_ANTRIEB_PRM";   // Becken 2 - ÜSS-Pumpe
      BB2_AS1 : "T_ANTRIEB_PRM";   // Becken 2 - Ablaufschieber 1
      BB2_AS2 : "T_ANTRIEB_PRM";   // Becken 2 - Ablaufschieber 2
      BB2_SR1 : "T_ANTRIEB_PRM";   // Becken 2 - MV Schlammrückführung 1
      BB2_SR2 : "T_ANTRIEB_PRM";   // Becken 2 - MV Schlammrückführung 2
      BB1_SR_K : "T_ANTRIEB_PRM";   // Becken 1- Druckluftkompressor Schlammrückführung
      Zulauf_AR_P1 : "T_ANTRIEB_PRM";   // Zulauf - Pumpwerk "Alter Rechen" - Pumpe 1
      Zulauf_AR_P2 : "T_ANTRIEB_PRM";   // Zulauf - Pumpwerk "Alter Rechen" - Pumpe 2
      Zulauf_AS : "T_ANTRIEB_PRM";   // Zulauf - Vorlagebehälter - Absperrschieber
      Zulauf_RA_SA : "T_ANTRIEB_PRM";   // Zulauf - Rechen - Sieb
      Zulauf_RA_HZS : "T_ANTRIEB_PRM";   // Zulauf - Rechen - HZS
      Zulauf_RA_VKS : "T_ANTRIEB_PRM";   // Zulauf - Rechen - VZS
      Zulauf_RA_V : "T_ANTRIEB_PRM";   // Zulauf - Rechen - Belüfter
      Zulauf_RA_RP : "T_ANTRIEB_PRM";   // Zulauf - Rechen - Räumpaddel
      Zulauf_RA_FP : "T_ANTRIEB_PRM";   // Zulauf - Rechen - Fettpumpe
      Schlamm_BP : "T_ANTRIEB_PRM";   // Schlamm - Beschickungspumpe Schlammbeete
      Truebwasser_P1 : "T_ANTRIEB_PRM";   // Trübwasserpumpwerk - Pumpe 1
      Truebwasser_P2 : "T_ANTRIEB_PRM";   // Trübwasserpumpwerk - Pumpe 2
      Schlamm_AS : "T_ANTRIEB_PRM";   // Schlamm - Absperrschieber Schlammbeete
      BB2_SR_K : "T_ANTRIEB_PRM";   // Becken 2 - Druckluftkompressor Schlammrückführung
      Zulauf_DosP : "T_ANTRIEB_PRM";   // Zulauf - Dosierpumpe
   END_STRUCT;


